# EPICS autosave request: hdf5App/Db/hdf5_settings.req
$(P)$(R)HDF5FilePath
$(P)$(R)HDF5Loop
$(P)$(R)HDF5AutoLoad
file "ADBase_settings.req", P=$(P), R=$(R)
